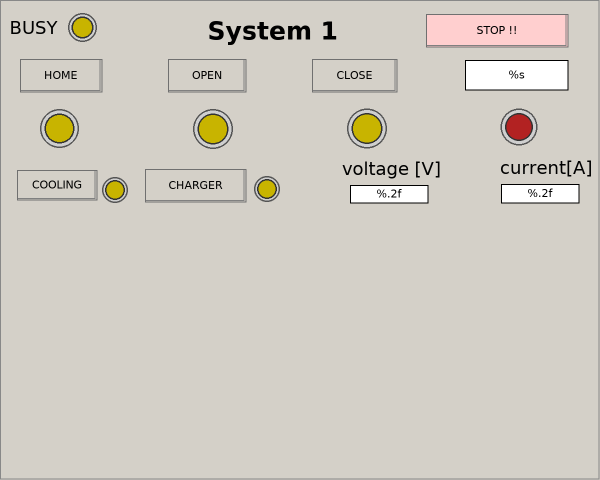
VISUALIZATION vACTION  // 600x480
VAR_IN_OUT
	vACTION:FB_ACTION;
	vACTION2:FB_ACTION;
END_VAR
    Button (20,59 82x33), "HOME", input disabled if: vACTION.bBUSY
        OnMouseDown: execute { vACTION.bHOME_ALL:=TRUE; }
    Lamp1 (37,103 45x51), variable: vACTION.bALL_HOMED, style: Lamp-Lamp1-Yellow
    Button (168,59 78x33), "OPEN", input disabled if: vACTION.bSAFE_MODE
        OnMouseDown: execute { vACTION.bOPEN_ALL:=TRUE; }
    Lamp1 (190,103 46x52), variable: vACTION.bALL_OPENED, style: Lamp-Lamp1-Yellow
    Button (312,59 85x33), "CLOSE", input disabled if: vACTION.bSAFE_MODE
        OnMouseDown: execute { vACTION.bCLOSE_ALL:=TRUE; }
    Lamp1 (344,103 46x51), variable: vACTION.bALL_CLOSED, style: Lamp-Lamp1-Yellow
    Lamp1 (498,104 42x46), variable: vACTION.bACTION_ERROR, style: Lamp-Lamp1-Red
    Rectangle (465,60 103x30), "%s", text variable: vACTION.sACTION_STATE
    Label (198,17 150x27), "System 1"
    Button (20,288 82x33), "HOME"
        OnMouseDown: execute { vACTION2.bHOME_ALL:=TRUE; }
    Lamp1 (37,332 45x51), variable: vACTION2.bALL_HOMED, style: Lamp-Lamp1-Yellow
    Button (168,288 78x33), "OPEN"
        OnMouseDown: execute { vACTION2.bOPEN_ALL:=TRUE; }
    Lamp1 (190,332 46x52), variable: vACTION2.bALL_OPENED, style: Lamp-Lamp1-Yellow
    Button (312,288 85x33), "CLOSE"
        OnMouseDown: execute { vACTION2.bCLOSE_ALL:=TRUE; }
    Lamp1 (344,332 46x51), variable: vACTION2.bALL_CLOSED, style: Lamp-Lamp1-Yellow
    Lamp1 (498,333 42x46), variable: vACTION2.bACTION_ERROR, style: Lamp-Lamp1-Red
    Rectangle (465,289 103x30), "%s", text variable: vACTION2.sACTION_STATE
    Label (121,252 150x30), "System 2"
    Button (145,169 101x33), "CHARGER"
        toggle vACTION.bCHARGE
    Rectangle (350,185 78x18), "%.2f", text variable: vACTION.iVOLTAGE_SHOW
    Label (339,155 105x28), "voltage [V]"
    Lamp1 (252,171 30x36), variable: vACTION.bCHARGE, style: Lamp-Lamp1-Yellow
    Button (16,391 101x33), "CHARGER ON"
        toggle vACTION2.bCHARGE
    Rectangle (286,391 103x30), "%f", text variable: vACTION2.iVOLTAGE_SHOW
    Label (155,396 150x30), "VOLTAGE:"
    Lamp1 (127,393 30x36), variable: vACTION2.bCHARGE, style: Lamp-Lamp1-Yellow
    Button (426,14 142x33), "STOP !!"
        OnMouseDown: execute { vACTION.bSTOP_ALL:=TRUE; }
    Button (428,249 140x33), "STOP !!"
        OnMouseDown: execute { vACTION.bSTOP_ALL:=TRUE; }
    Rectangle (7,240 571x227), invisible if: bSECOND_SYS
    Lamp1 (66,10 33x35), variable: LED, style: Lamp-Lamp1-Yellow
    Label (-5,13 77x30), "BUSY"
    Label (498,153 97x30), "current[A]"
    Rectangle (501,184 78x19), "%.2f", text variable: vACTION.iCURRENT_CHARGE_SHOW
    Button (17,170 80x30), "COOLING"
        toggle ACTION1.bPTC_ON
    Lamp1 (100,172 30x36), variable: PTCon, style: Lamp-Lamp1-Yellow
END_VISUALIZATION

(* stored: Version 1.1.0.1, ProductVersion 3.1.4024.12
   Visu vACTION: Id {d21375e2-c764-44f8-9c50-3c770c1388ac} *)
